Yaskawa INFORM job: TWFUFGET.JBI

/JOB
//NAME TWFUFGET
//POS
///NPOS 0,0,0,0,0,0
//INST
///DATE 2024/04/10 14:36
///ATTR SC,RW
///GROUP1 RB1,BS1
NOP
SETTM TM000 TRESET
SETTM TM000 TSTART
TIMER T=5.00
PAUSE
TIMER T=5.00
SETTM TM000 TSTOP
END
